PROGRAM FUN_CompressCSV
VAR_INPUT
	InDirectory 		: T_MaxString;
END_VAR
VAR_OUTPUT
END_VAR
VAR
	Directory1		: T_MaxString;
	Directory2		: T_MaxString;
	FB_Time 			: FB_LocalSystemTime;
	CompressFile	: FB_CompressFile;
	PreviousMonth 	: WORD := 12;
	PreviousYear 	: WORD := 2018;
	CalDirectory 	: T_MaxString;
	DirChange		: BOOL;
	bTest 			: BOOL;
	TimeStruct_Local : TIMESTRUCT;
END_VAR

FB_Time(sNetID := '', bEnable := TRUE, dwCycle := 1, dwOpt := 1, tTimeout := T#50MS, systemTime => TimeStruct_Local);
IF FB_TIME.bValid THEN 
	IF PreviousMonth <> TimeStruct_Local.wMonth THEN
		Directory1 := Concat(InDirectory, concat(WORD_TO_STRING(TimeStruct_Local.wYear), '\'));
		
		IF PreviousYear <> TimeStruct_Local.wYear THEN
			Directory1 := Concat(InDirectory, concat(WORD_TO_STRING(TimeStruct_Local.wYear-1), '\'));
			PreviousYear := TimeStruct_Local.wYear;
		END_IF
		
		Directory2 := Concat(Directory1, concat(WORD_TO_STRING(PreviousMonth), '\'));
		PreviousMonth := TimeStruct_Local.wMonth;
		DirChange := TRUE;
	END_IF

	
	IF DirChange THEN	
		bTest := TRUE;
		CompressFile(IN_Directory := Directory2);	
		DirChange := FALSE;
	END_IF
END_IF

END_PROGRAM

(* stored: Version 1.1.0.1, ProductVersion 3.1.4024.6
   POU FUN_CompressCSV: Id {569cc088-ec71-40f8-bf76-c21db6198aa5}, SpecialFunc None *)
